// TIA Portal project "plc-proje-sim" (V15.1)

(* hardware
DEVICE "S71500/ET200MP-Station_1"  S7-1500 station
   slot 0: "Profilschiene_0"  6ES7 590-1***0-0AA0
   slot 1: "PLC_1"  CPU 1511-1 PN  6ES7 511-1AK00-0AB0  V1.8
   slot 2: "AI 8xU/I/RTD/TC ST_1"  AI 8xU/I/RTD/TC ST  6ES7 531-7KF00-0AB0  V2.0
   slot 3: "AI 8xU/I/RTD/TC ST_2"  AI 8xU/I/RTD/TC ST  6ES7 531-7KF00-0AB0  V2.0
   slot 4: "AI 8xU/I/RTD/TC ST_3"  AI 8xU/I/RTD/TC ST  6ES7 531-7KF00-0AB0  V2.0
   slot 5: "AI 8xU/I/RTD/TC ST_4"  AI 8xU/I/RTD/TC ST  6ES7 531-7KF00-0AB0  V2.0
   slot 6: "DI 16x24VDC BA_1"  DI 16x24VDC BA  6ES7 521-1BH10-0AA0  V1.0
*)

// ===== PLC "PLC_1"  CPU 1511-1 PN =====

VAR_GLOBAL   // PLC tag table "Standard-Variablentabelle"
   "ACIL" AT %I0.2 : Bool;
   "start" AT %I0.0 : Bool;
   "stop" AT %I0.1 : Bool;
   "sistem" AT %M0.0 : Bool;
   "düsük konveyor" AT %QW30 : Word;
   "orta konveyor" AT %QW32 : Word;
   "yuksek konveyor" AT %QW34 : Word;
   "DUSUK GOSTERGE DISPLAY" AT %QW40 : Word;
   "ORTA GOSTERGE DISPLAY" AT %QW42 : Word;
   "YUKSEK GOTERGE DISPLAY" AT %QW44 : Word;
   "AGIRLIK ANLIK" AT %QW38 : Word;
   "TEMP2" AT %MD110 : Real;
   "AGIRLIK KON INPUT" AT %IW32 : Word;
   "ANA KONVEYOR" AT %QW46 : Word;
   "TEMP 3" AT %MD120 : Real;
   "Tag_5" AT %MW48 : Int;
   "Tag_6" AT %MW50 : Int;
   "DUSUK SENSOR" AT %I0.3 : Bool;
   "ORTA SENSOR" AT %I0.4 : Bool;
   "YUKSEK SENSOR" AT %I0.5 : Bool;
   "AGIRLIK SENSOR" AT %I0.7 : Bool;
   "RESET TUSU" AT %I0.6 : Bool;
   "AGIRLIK KONVEYORU" AT %Q1.0 : Bool;
   "SAG DUSUK KONVEYOR" AT %Q1.2 : Bool;
   "SOL ORTA KONVEYOR" AT %Q1.3 : Bool;
   "DUZ BUYUK KONVEYOR" AT %Q1.4 : Bool;
   "HIZ GOSTERGESI DISPLAY" AT %QW36 : Word;
   "potansıyometre" AT %IW30 : Word;
   "TEMP1" AT %MD100 : DWord;
   "TEMP 4" AT %MD200 : DWord;
   "TOPLAM KUTU SAYISI" AT %MW52 : Int;
END_VAR

// folder: System blocks/Program resources

DATA_BLOCK "IEC_Counter_0_DB_DUSUK"   // DB1
{ S7_Optimized_Access := 'TRUE' }
AUTHOR : Simatic
FAMILY : IEC
NAME : CNTR
VERSION : 1.0
// stored: InstanceOfName IEC_COUNTER
"IEC_COUNTER"
BEGIN
END_DATA_BLOCK

DATA_BLOCK "IEC_Counter_0_DB_ORTA"   // DB2
{ S7_Optimized_Access := 'TRUE' }
AUTHOR : Simatic
FAMILY : IEC
NAME : CNTR
VERSION : 1.0
// stored: InstanceOfName IEC_COUNTER
"IEC_COUNTER"
BEGIN
END_DATA_BLOCK

DATA_BLOCK "IEC_Counter_0_DB_YUKSEK"   // DB3
{ S7_Optimized_Access := 'TRUE' }
AUTHOR : Simatic
FAMILY : IEC
NAME : CNTR
VERSION : 1.0
// stored: InstanceOfName IEC_COUNTER
"IEC_COUNTER"
BEGIN
END_DATA_BLOCK

DATA_BLOCK "IEC_Timer_0_DB_AGIRLIK_KON"   // DB4
{ S7_Optimized_Access := 'TRUE' }
AUTHOR : Simatic
FAMILY : IEC
NAME : IEC_TMR
VERSION : 1.0
// stored: InstanceOfName IEC_TIMER
"IEC_TIMER"
BEGIN
END_DATA_BLOCK

DATA_BLOCK "IEC_Timer_0_DB"   // DB5
{ S7_Optimized_Access := 'TRUE' }
AUTHOR : Simatic
FAMILY : IEC
NAME : IEC_TMR
VERSION : 1.0
// stored: InstanceOfName IEC_TIMER
"IEC_TIMER"
BEGIN
END_DATA_BLOCK

DATA_BLOCK "IEC_Timer_0_DB_1"   // DB6
{ S7_Optimized_Access := 'TRUE' }
AUTHOR : Simatic
FAMILY : IEC
NAME : IEC_TMR
VERSION : 1.0
// stored: InstanceOfName IEC_TIMER
"IEC_TIMER"
BEGIN
END_DATA_BLOCK

DATA_BLOCK "IEC_Timer_0_DB_2"   // DB7
{ S7_Optimized_Access := 'TRUE' }
AUTHOR : Simatic
FAMILY : IEC
NAME : IEC_TMR
VERSION : 1.0
// stored: InstanceOfName IEC_TIMER
"IEC_TIMER"
BEGIN
END_DATA_BLOCK

DATA_BLOCK "IEC_Timer_0_DB_3"   // DB8
{ S7_Optimized_Access := 'TRUE' }
AUTHOR : Simatic
FAMILY : IEC
NAME : IEC_TMR
VERSION : 1.0
// stored: InstanceOfName IEC_TIMER
"IEC_TIMER"
BEGIN
END_DATA_BLOCK

// folder: (top level)

FUNCTION "MHJ-PLC-Lab-Function-S71500" : Void   // FC9000, SCL
{ S7_Optimized_Access := 'TRUE' }
VERSION : 0.1
   VAR_TEMP
      Value : Byte;
      ForCounter : Int;
   END_VAR
   VAR CONSTANT
      Value_01_DW : DWord := 16#1223_5486;
      Value_02_DW : DWord := 16#A6C9_D1F5;
   END_VAR
BEGIN

   #Value:=PEEK(area := 16#82,
        dbNumber := 0,
        byteOffset := 511);
   #Value := #Value + 1;

   POKE(area := 16#82,
        dbNumber := 0,
        byteOffset := 511,
        value := #Value);

   POKE(area := 16#82,
        dbNumber := 0,
        byteOffset := 1016,
        value := #Value_01_DW);
   POKE(area := 16#82,
        dbNumber := 0,
        byteOffset := 1020,
        value := #Value_02_DW);

   FOR #ForCounter := 0 TO 63 DO
       #Value:=PEEK(area := 16#1,
            dbNumber := 0,
            byteOffset := #ForCounter);
       POKE(area := 16#81,
            dbNumber := 0,
            byteOffset := #ForCounter,
            value := #Value);
   END_FOR;
   #Value := PEEK(area := 16#1,
                  dbNumber := 0,
                  byteOffset := 512);
   POKE(area := 16#82,
        dbNumber := 0,
        byteOffset := 512,
        value := #Value);
END_FUNCTION

ORGANIZATION_BLOCK "Main"   // OB1, LAD, ProgramCycle
TITLE = "Main Program Sweep (Cycle)"
{ S7_Optimized_Access := 'TRUE' }
VERSION : 0.1
   VAR_INPUT
      Initial_Call : Bool;   // Initial call of this OB
      Remanence : Bool;   // =True, if remanent data are available
   END_VAR
   VAR_TEMP   // added for the SCL form of the ladder/FBD networks
      _w1 : Bool;
      _w2 : Bool;
      _w3 : Bool;
   END_VAR
BEGIN

REGION Network 1
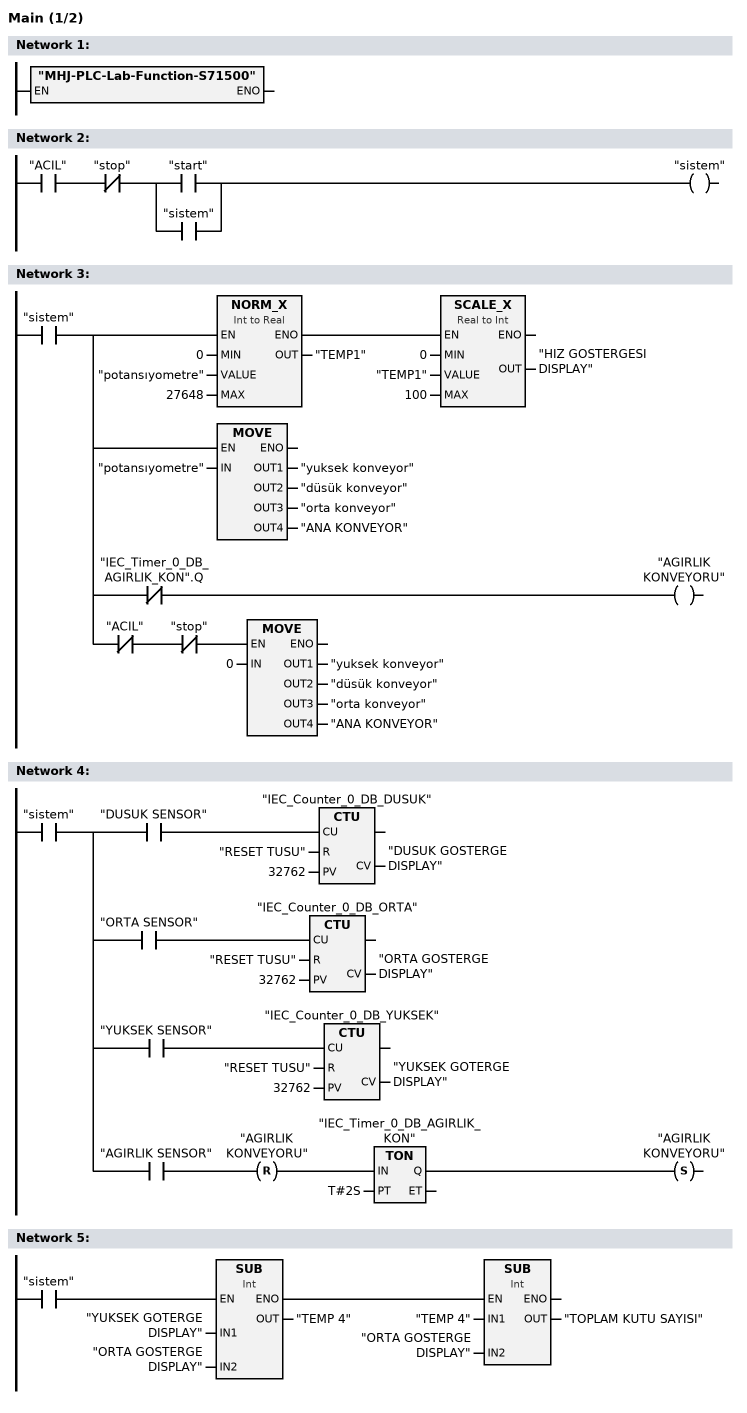
   RUNG wire#powerrail
      "MHJ-PLC-Lab-Function-S71500"()
   END_RUNG
   // the same network as SCL:
   "MHJ-PLC-Lab-Function-S71500"();
END_REGION

REGION Network 2
   RUNG wire#powerrail
      Contact( "ACIL" )
      I_Contact( "stop" )
      wire#w1
      Contact( "start" )
      wire#w2
      Coil( "sistem" )
   END_RUNG
   RUNG wire#w1
      Contact( "sistem" )
   END_RUNG wire#w2
   // the same network as SCL:
   "sistem" := "ACIL" AND NOT "stop" AND ("start" OR "sistem");
END_REGION

REGION Network 3
   RUNG wire#powerrail
      Contact( "sistem" )
      wire#w1
      { S7_Templates := "[SrcType := Int, DestType := Real]" } Normalize(min := 0, value := "potansıyometre", max := 27648, out => "TEMP1")
      { S7_Templates := "[SrcType := Real, DestType := Int]" } Scale(min := 0, value := "TEMP1", max := 100, out => "HIZ GOSTERGESI DISPLAY")
   END_RUNG
   RUNG wire#w1
      Move(in := "potansıyometre", out1 => "yuksek konveyor", out2 => "düsük konveyor", out3 => "orta konveyor", out4 => "ANA KONVEYOR")
   END_RUNG
   RUNG wire#w1
      I_Contact( "IEC_Timer_0_DB_AGIRLIK_KON".Q )
      Coil( "AGIRLIK KONVEYORU" )
   END_RUNG
   RUNG wire#w1
      I_Contact( "ACIL" )
      I_Contact( "stop" )
      Move(in := 0, out1 => "yuksek konveyor", out2 => "düsük konveyor", out3 => "orta konveyor", out4 => "ANA KONVEYOR")
   END_RUNG
   // the same network as SCL:
   IF "sistem" THEN
       "TEMP1" := NORM_X(MIN := 0, VALUE := "potansıyometre", MAX := 27648);
       "HIZ GOSTERGESI DISPLAY" := SCALE_X(MIN := 0, VALUE := "TEMP1", MAX := 100);
       "yuksek konveyor" := "potansıyometre";
       "düsük konveyor" := "potansıyometre";
       "orta konveyor" := "potansıyometre";
       "ANA KONVEYOR" := "potansıyometre";
   END_IF;
   "AGIRLIK KONVEYORU" := "sistem" AND NOT "IEC_Timer_0_DB_AGIRLIK_KON".Q;
   IF "sistem" AND NOT "ACIL" AND NOT "stop" THEN
       "yuksek konveyor" := 0;
       "düsük konveyor" := 0;
       "orta konveyor" := 0;
       "ANA KONVEYOR" := 0;
   END_IF;
END_REGION

REGION Network 4
   "IEC_Counter_0_DB_DUSUK".CTU(CU := "sistem" AND "DUSUK SENSOR",
                           R := "RESET TUSU",
                           PV := 32762,
                           CV => "DUSUK GOSTERGE DISPLAY");
   "IEC_Counter_0_DB_ORTA".CTU(CU := "sistem" AND "ORTA SENSOR",
                           R := "RESET TUSU",
                           PV := 32762,
                           CV => "ORTA GOSTERGE DISPLAY");
   "IEC_Counter_0_DB_YUKSEK".CTU(CU := "sistem" AND "YUKSEK SENSOR",
                           R := "RESET TUSU",
                           PV := 32762,
                           CV => "YUKSEK GOTERGE DISPLAY");
   #_w1 := "sistem" AND "AGIRLIK SENSOR";
   IF #_w1 THEN "AGIRLIK KONVEYORU" := FALSE; END_IF;
   "IEC_Timer_0_DB_AGIRLIK_KON".TON(IN := #_w1, PT := T#2S);
   IF "IEC_Timer_0_DB_AGIRLIK_KON".Q THEN "AGIRLIK KONVEYORU" := TRUE; END_IF;
END_REGION

REGION Network 5
   RUNG wire#powerrail
      Contact( "sistem" )
      { S7_Templates := "SrcType := Int" } Sub(in1 := "YUKSEK GOTERGE DISPLAY", in2 := "ORTA GOSTERGE DISPLAY", out => "TEMP 4")
      { S7_Templates := "SrcType := Int" } Sub(in1 := "TEMP 4", in2 := "ORTA GOSTERGE DISPLAY", out => "TOPLAM KUTU SAYISI")
   END_RUNG
   // the same network as SCL:
   IF "sistem" THEN
       "TEMP 4" := "YUKSEK GOTERGE DISPLAY" - "ORTA GOSTERGE DISPLAY";
       "TOPLAM KUTU SAYISI" := "TEMP 4" - "ORTA GOSTERGE DISPLAY";
   END_IF;
END_REGION

REGION Network 6
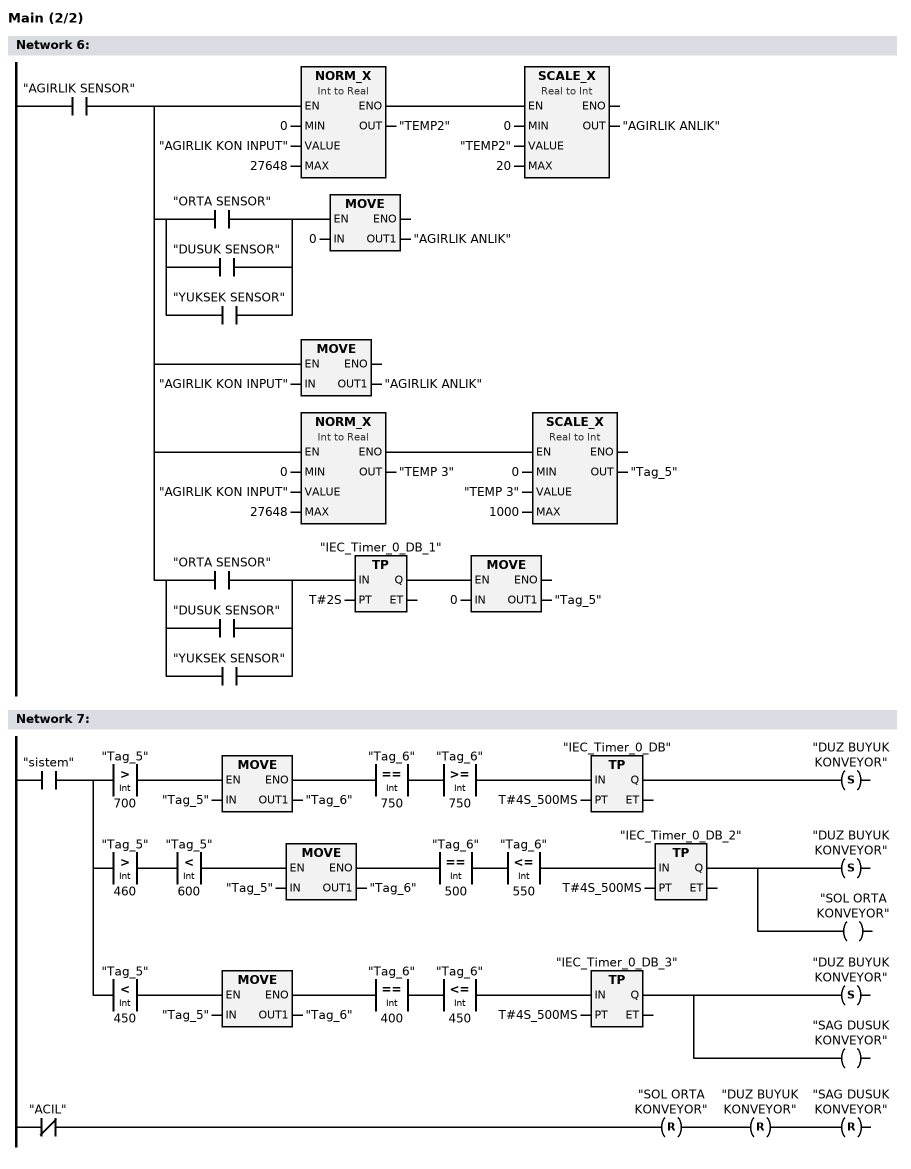
   IF "AGIRLIK SENSOR" THEN
       "TEMP2" := NORM_X(MIN := 0, VALUE := "AGIRLIK KON INPUT", MAX := 27648);
       "AGIRLIK ANLIK" := SCALE_X(MIN := 0, VALUE := "TEMP2", MAX := 20);
   END_IF;
   IF "AGIRLIK SENSOR" AND ("ORTA SENSOR" OR "DUSUK SENSOR" OR "YUKSEK SENSOR") THEN
       "AGIRLIK ANLIK" := 0;
   END_IF;
   IF "AGIRLIK SENSOR" THEN
       "AGIRLIK ANLIK" := "AGIRLIK KON INPUT";
       "TEMP 3" := NORM_X(MIN := 0, VALUE := "AGIRLIK KON INPUT", MAX := 27648);
       "Tag_5" := SCALE_X(MIN := 0, VALUE := "TEMP 3", MAX := 1000);
   END_IF;
   "IEC_Timer_0_DB_1".TP(IN := "AGIRLIK SENSOR" AND ("ORTA SENSOR" OR "DUSUK SENSOR" OR "YUKSEK SENSOR"),
                         PT := T#2S);
   IF "IEC_Timer_0_DB_1".Q THEN "Tag_5" := 0; END_IF;
END_REGION

REGION Network 7
   #_w1 := "sistem" AND ("Tag_5" > 700);
   IF #_w1 THEN "Tag_6" := "Tag_5"; END_IF;
   "IEC_Timer_0_DB".TP(IN := #_w1 AND ("Tag_6" = 750) AND ("Tag_6" >= 750), PT := T#4S_500MS);
   IF "IEC_Timer_0_DB".Q THEN "DUZ BUYUK KONVEYOR" := TRUE; END_IF;
   #_w2 := "sistem" AND ("Tag_5" > 460) AND ("Tag_5" < 600);
   IF #_w2 THEN "Tag_6" := "Tag_5"; END_IF;
   "IEC_Timer_0_DB_2".TP(IN := #_w2 AND ("Tag_6" = 500) AND ("Tag_6" <= 550), PT := T#4S_500MS);
   IF "IEC_Timer_0_DB_2".Q THEN "DUZ BUYUK KONVEYOR" := TRUE; END_IF;
   "SOL ORTA KONVEYOR" := "IEC_Timer_0_DB_2".Q;
   #_w3 := "sistem" AND ("Tag_5" < 450);
   IF #_w3 THEN "Tag_6" := "Tag_5"; END_IF;
   "IEC_Timer_0_DB_3".TP(IN := #_w3 AND ("Tag_6" = 400) AND ("Tag_6" <= 450), PT := T#4S_500MS);
   IF "IEC_Timer_0_DB_3".Q THEN "DUZ BUYUK KONVEYOR" := TRUE; END_IF;
   "SAG DUSUK KONVEYOR" := "IEC_Timer_0_DB_3".Q;
   IF NOT "ACIL" THEN
       "SOL ORTA KONVEYOR" := FALSE;
       "DUZ BUYUK KONVEYOR" := FALSE;
       "SAG DUSUK KONVEYOR" := FALSE;
   END_IF;
END_REGION
END_ORGANIZATION_BLOCK